{attribute addProperty BoxType "EJ7037-0000-0020"}
{attribute addProperty Id "ControlAT %Q*Control_D763B957162"}
{attribute addProperty CRC "2448212702"}
{attribute addProperty SizeInBites "16"}
{attribute addProperty SizeInBytes "2"}
TYPE STM_Control_91ECC2DE :
STRUCT
	{attribute addProperty Name "Control"}
	Control AT %Q* : Control_D763B957;
END_STRUCT
END_TYPE

(* stored: Version 1.2.0.0, ProductVersion 3.1.4024.9
   DUT STM_Control_91ECC2DE: Id {ea6f5131-5468-4e95-afa5-a9e3cf200ea5} *)
